{attribute addProperty BoxType "KL1501"}
{attribute addProperty Id "StateAT %I*USINT000Data_InAT %I*ARRAY [0..1] OF UINT000CtrlAT %Q*USINT000Data_OutAT %Q*ARRAY [0..1] OF UINT000"}
{attribute addProperty CRC "3378628486"}
{attribute addProperty SizeInBites "0"}
{attribute addProperty SizeInBytes "0"}
TYPE Channel_C961C786 :
STRUCT
	{attribute addProperty Name "State"}
	State AT %I* : USINT;
	{attribute addProperty Name "Data_In"}
	Data_In AT %I* : ARRAY [0..1] OF UINT;
	{attribute addProperty Name "Ctrl"}
	Ctrl AT %Q* : USINT;
	{attribute addProperty Name "Data_Out"}
	Data_Out AT %Q* : ARRAY [0..1] OF UINT;
END_STRUCT
END_TYPE

(* stored: Version 1.2.0.0, ProductVersion 3.1.4024.9
   DUT Channel_C961C786: Id {a44ca60c-2c8a-4007-86e2-211792fb5669} *)
